TYPE ST_MBM_IO :
STRUCT
	stHwInMbm		AT%I*	: ST_Euchner_MBM_HW_IN;
	stHwOutMbm		AT%Q*	: ST_Euchner_MBM_HW_OUT;
END_STRUCT
END_TYPE

(* stored: Version 1.1.0.1, ProductVersion 3.1.4024.12
   DUT ST_MBM_IO: Id {69dd27f3-994c-41e6-ac6b-5ccd722a8936} *)
